FUNCTION_BLOCK TESTER (* Test wrapper for IEC 61131-3 FBs *)
  (* Standard: 61499-1 *)
  (* Version 0.0, 2000-02-13, JHC, Rockwell Automation, Replacement for lost source *)
  (* Compiler header: package fb.rt.hmi; *)
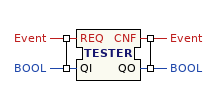
  EVENT_INPUT
    REQ WITH QI; (* Normal Execution Request *)
  END_EVENT
  EVENT_OUTPUT
    CNF WITH QO; (* Execution Confirmation *)
  END_EVENT
  VAR_INPUT
    QI : BOOL; (* Input event qualifier *)
  END_VAR
  VAR_OUTPUT
    QO : BOOL; (* Output event qualifier *)
  END_VAR
END_FUNCTION_BLOCK
